FUNCTION_BLOCK AxisFunctionBlocks
VAR_IN_OUT
	Axis					:AXIS_REF;	
	Control					:CTR_SIGNALS_INTERNAL;
	Output					:OUT_SIGNALS;
	HomeStatus				:MOTION_FB_STATUS;
END_VAR	
VAR
	//function blocks
	mcPower					:MC_Power;
	mcSetPosition			:MC_SetPosition;
	mcMoveAbsolute			:MC_MoveAbsolute;
	mcMoveRelative			:MC_MoveRelative;
	mcMoveVelocity			:MC_MoveVelocity;
	mcReset					:MC_Reset;
	mcHalt					:MC_Halt;
	mcStop					:MC_Stop;
	mcReadActualVelocity	:MC_ReadActualVelocity;
	mcReadActualPosition	:MC_ReadActualPosition;
	mcJog					:MC_Jog;
	mcHome					:MC_Home;	
	mcGearIn				:MC_GearIn;
	mcGearOut				:MC_GearOut;
END_VAR
VAR // added by the converter: edge detectors and wires of the graphical bodies
    _w1, _w5, _w6, _w8, _w11 : BOOL;
    _w2, _w3, _w4, _w7, _w9, _w10 : ANY;
END_VAR

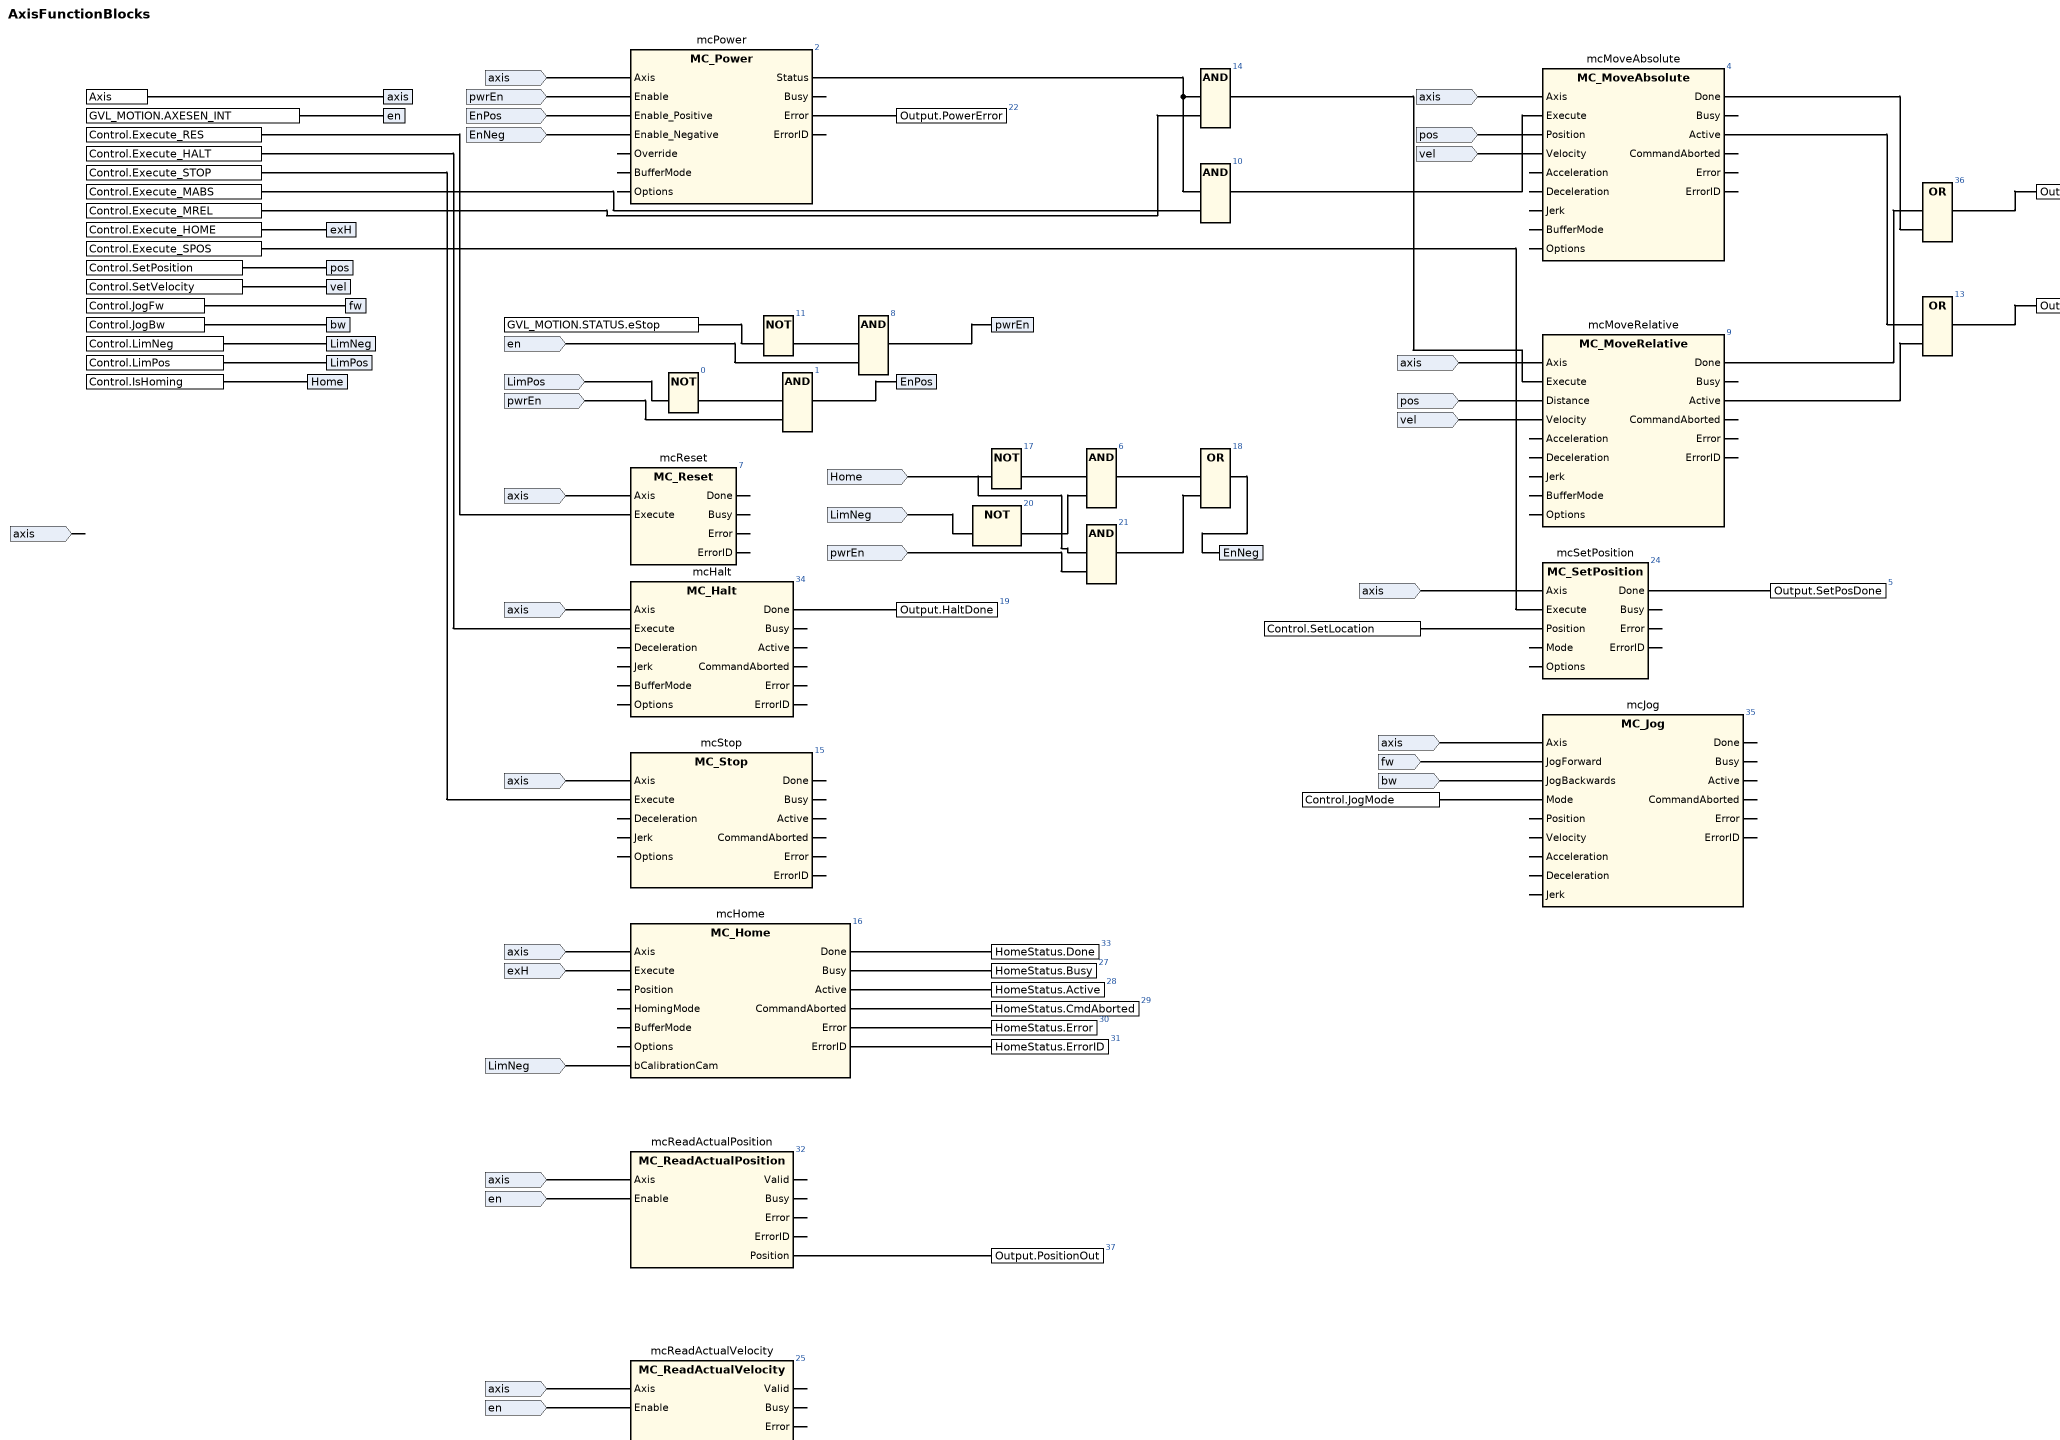
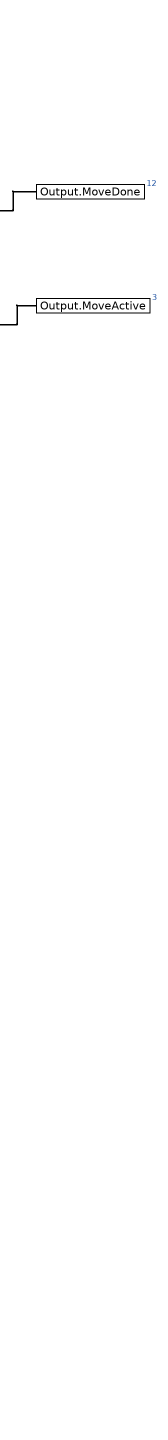
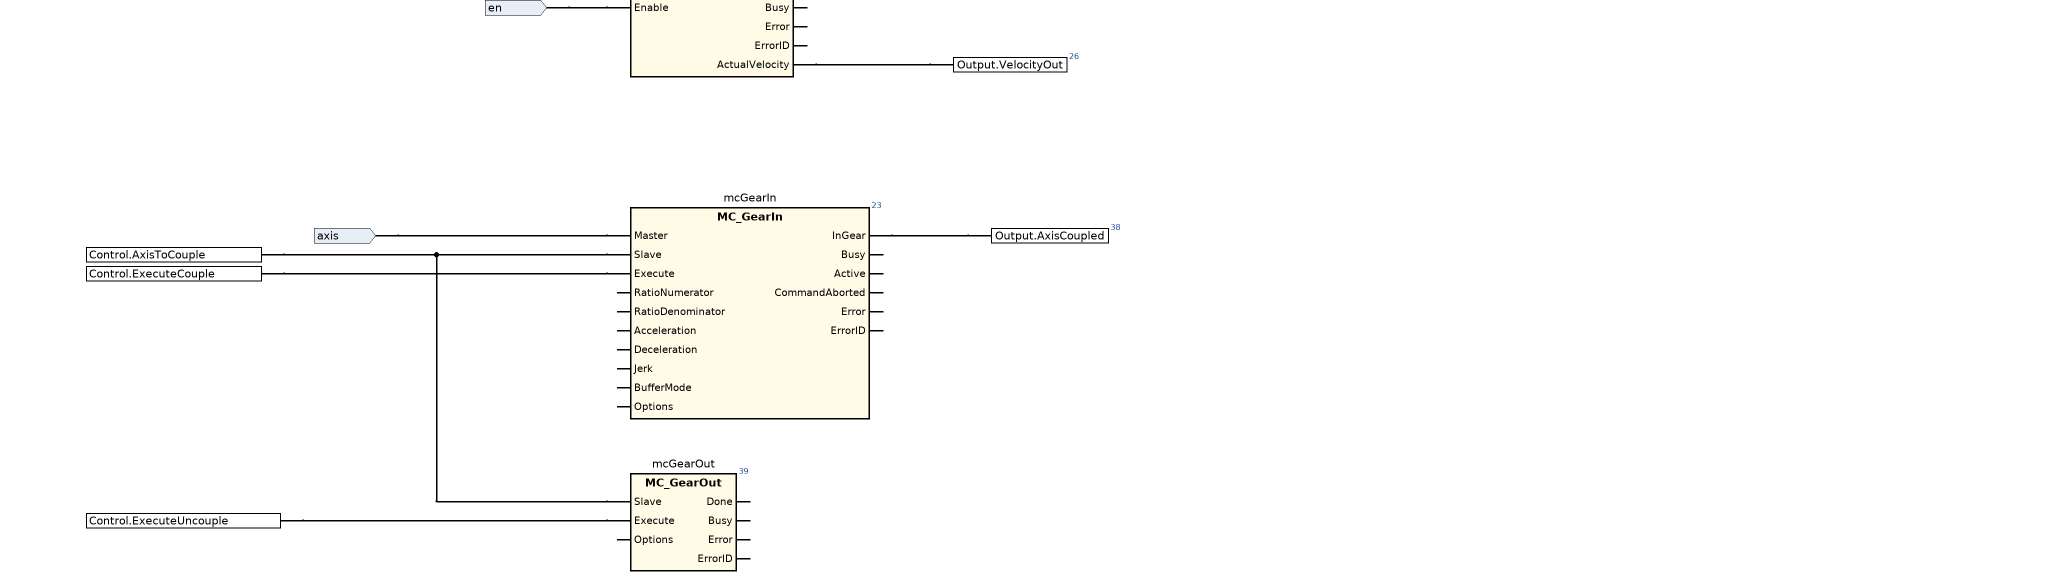
mcPower(Axis := Axis, Enable := _w1, Enable_Positive := NOT Control.LimPos AND _w1, Enable_Negative := _w2); // MC_Power
Output.MoveActive := _w3;
mcMoveAbsolute(
    Axis := Axis,
    Execute := _w4,
    Position := Control.SetPosition,
    Velocity := Control.SetVelocity); // MC_MoveAbsolute
Output.SetPosDone := mcSetPosition.Done;
_w7 := _w5 AND _w6;
mcReset(Axis := Axis, Execute := Control.Execute_RES); // MC_Reset
_w1 := _w8 AND GVL_MOTION.AXESEN_INT;
mcMoveRelative(
    Axis := Axis,
    Execute := _w9,
    Distance := Control.SetPosition,
    Velocity := Control.SetVelocity); // MC_MoveRelative
_w4 := mcPower.Status AND Control.Execute_MABS;
_w8 := NOT GVL_MOTION.STATUS.eStop;
Output.MoveDone := _w10;
_w3 := mcMoveAbsolute.Active OR mcMoveRelative.Active;
_w9 := mcPower.Status AND Control.Execute_MREL;
mcStop(Axis := Axis, Execute := Control.Execute_STOP); // MC_Stop
mcHome(Axis := Axis, Execute := Control.Execute_HOME, bCalibrationCam := Control.LimNeg); // MC_Home
_w5 := NOT Control.IsHoming;
_w2 := _w7 OR _w11;
Output.HaltDone := mcHalt.Done;
_w6 := NOT Control.LimNeg;
_w11 := Control.IsHoming AND _w1;
Output.PowerError := mcPower.Error;
mcGearIn(Master := Axis, Slave := Control.AxisToCouple, Execute := Control.ExecuteCouple); // MC_GearIn
mcSetPosition(Axis := Axis, Execute := Control.Execute_SPOS, Position := Control.SetLocation); // MC_SetPosition
mcReadActualVelocity(Axis := Axis, Enable := GVL_MOTION.AXESEN_INT); // MC_ReadActualVelocity
Output.VelocityOut := mcReadActualVelocity.ActualVelocity;
HomeStatus.Busy := mcHome.Busy;
HomeStatus.Active := mcHome.Active;
HomeStatus.CmdAborted := mcHome.CommandAborted;
HomeStatus.Error := mcHome.Error;
HomeStatus.ErrorID := mcHome.ErrorID;
mcReadActualPosition(Axis := Axis, Enable := GVL_MOTION.AXESEN_INT); // MC_ReadActualPosition
HomeStatus.Done := mcHome.Done;
mcHalt(Axis := Axis, Execute := Control.Execute_HALT); // MC_Halt
mcJog(Axis := Axis, JogForward := Control.JogFw, JogBackwards := Control.JogBw, Mode := Control.JogMode); // MC_Jog
_w10 := mcMoveRelative.Done OR mcMoveAbsolute.Done;
Output.PositionOut := mcReadActualPosition.Position;
Output.AxisCoupled := mcGearIn.InGear;
mcGearOut(Slave := Control.AxisToCouple, Execute := Control.ExecuteUncouple); // MC_GearOut

END_FUNCTION_BLOCK

(* stored: Version 1.1.0.1, ProductVersion 3.1.4026.18
   POU AxisFunctionBlocks: Id {97c0c113-3b4a-4576-88ff-a16c0cbb43a0}, SpecialFunc None *)
